FUNCTION_BLOCK ProcessDataManager EXTENDS TcoData.TcoDataExchange
VAR
	//this variable has to called "_data" - PC app will access this variable by its name.
	_data : Station001_ProductionData;
END_VAR

SUPER^();

END_FUNCTION_BLOCK

(* stored: Version 1.1.0.1, ProductVersion 3.1.4024.9
   POU ProcessDataManager: Id {ef58d043-6bbe-480b-9350-92a4de31085d}, SpecialFunc None *)
